FUNCTION F_TrackSettingChangesWs : BOOL
VAR_INPUT
	sValue		: WSTRING;
END_VAR
VAR_IN_OUT
	stSetting	: ST_Data_Item;
	sChanges	: STRING;
END_VAR

IF stSetting.sValue <> sValue THEN
	sChanges := Concat7(sChanges, '$N ', WSTRING_TO_STRING(stSetting.stName.wsName), ' ', TO_STRING(stSetting.sValue), ' -> ', TO_STRING(sValue));
END_IF

stSetting.sValue := sValue;
F_TrackSettingChangesWs := TRUE;

END_FUNCTION

(* stored: Version 1.1.0.1, ProductVersion 3.1.4024.12
   POU F_TrackSettingChangesWs: Id {180d96da-508f-4f9e-b8fc-cc11bf2f478f}, SpecialFunc None *)
